(* IEC 61131-3 sources: plc_on_fpga_riscv_hybrid/RV_FPGA_PLC_IDE_Projects/Arithmatic, 1 file *)

(* ---- Arithmatic.il ---- *)
VAR
    Add_Res   : INT
END_VAR

PROGRAM Arithmatic
    Addition :
        LD     25
        ADD    16
        ST     Add_Res
    Check_Res :
        LD     Add_Res
        EQ     41
        ST     %LEDG.0
    Check_Error :
        LD     Add_Res
        NE     41
        ST     %LEDR.0
    Check_2 :
        LD     Add_Res
        LT     50
        ST     %LEDG.7
END_PROGRAM
